VAR_GLOBAL
	Null:			PVOID:= 0;
END_VAR

(* stored: Version 1.1.0.1, ProductVersion 3.1.4024.12
   GVL GVL: Id {ecdb87fb-27ae-4e70-b884-18b66c1ba2c5} *)
